Staubli VAL3: setValue.pgx

public program setValue(num& x_nValue[], string x_sItem)
begin
  if find(x_sItem,"In")==-1
    // set the data only for output
    if isDefined(saveInOut:cCount[x_sItem])
      saveInOut:cCount[x_sItem].nCount=x_nValue
    elseIf isDefined(saveInOut:aCount[x_sItem])
      aioSet(saveInOut:aCount[x_sItem].aAio,x_nValue)
    endIf
  endIf
end
